INTERFACE ACDCChargerElement

METHOD Disable : BOOL
VAR_INPUT
END_VAR
END_METHOD

METHOD Enable : BOOL
VAR_INPUT
END_VAR
END_METHOD

METHOD SetPowerLevel : BOOL
VAR_INPUT
END_VAR
END_METHOD

END_INTERFACE

(* stored: Version 1.1.0.1, ProductVersion 3.1.4024.12
   Itf ACDCChargerElement: Id {7d70f492-a55e-4bd4-9bfa-0d7b80bc7086}
   Method Disable: Id {fc171ec4-5a66-4524-b0da-65c411c7cf1f}
   Method Enable: Id {22c8f2cf-3020-4447-8555-6a828de5b146}
   Method SetPowerLevel: Id {7a5b812d-c068-4973-b22c-954f88eb422c} *)
